// TIA Portal V17 export
FUNCTION "FC_风机燃气控制" : Void   // FC, LAD
{ S7_Optimized_Access := 'TRUE' }
   VAR_TEMP
      风机控制输出值 : Real;
      风压过渡 : Int;
   END_VAR
BEGIN

REGION Network 1: 风机运行控制
   // 常开触点风机运行按与常闭触点风机故障反馈串联，当风机运行按接通且风机故障反馈未动作时，驱动风机运行线圈Q4.4
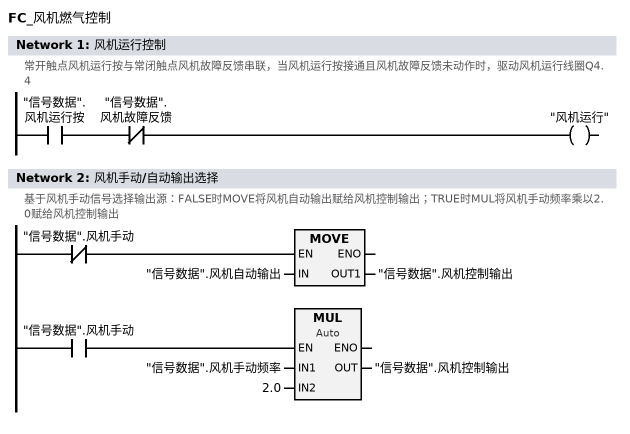
   RUNG wire#powerrail
      Contact( "信号数据".风机运行按 )
      I_Contact( "信号数据".风机故障反馈 )
      Coil( "风机运行" )
   END_RUNG
   // the same network as SCL:
   "风机运行" := "信号数据".风机运行按 AND NOT "信号数据".风机故障反馈;
END_REGION

REGION Network 2: 风机手动/自动输出选择
   // 基于风机手动信号选择输出源：FALSE时MOVE将风机自动输出赋给风机控制输出；TRUE时MUL将风机手动频率乘以2.0赋给风机控制输出
   RUNG wire#powerrail
      I_Contact( "信号数据".风机手动 )
      { S7_GenerateENO := "TRUE" } Move(in := "信号数据".风机自动输出, out1 => "信号数据".风机控制输出)
   END_RUNG
   RUNG wire#powerrail
      Contact( "信号数据".风机手动 )
      { S7_GenerateENO := "TRUE" } Mul(in1 := "信号数据".风机手动频率, in2 := 2.0, out => "信号数据".风机控制输出)
   END_RUNG
   // the same network as SCL:
   IF NOT "信号数据".风机手动 THEN "信号数据".风机控制输出 := "信号数据".风机自动输出; END_IF;
   IF "信号数据".风机手动 THEN "信号数据".风机控制输出 := "信号数据".风机手动频率 * 2.0; END_IF;
END_REGION
END_FUNCTION
